FUNCTION_BLOCK FB_Encoder
VAR_INPUT
	nRawInput : UDINT;
	fEncoderOffset : LREAL; 
END_VAR
VAR_OUTPUT
	fPosition 		: LREAL;
	fPositionError 	: LREAL;
END_VAR
VAR PERSISTENT
	nRounds			: DINT;
	nRawLast 		: DINT;
END_VAR	
VAR
	nInput 		: DINT;
	nTempInputDiff	: DINT;
	nCount 			: DINT;
	nMaxValue30bit 	: DINT :=  1073741823; // 2^30 - 1	
	nThreshold30bit	: DINT := nMaxValue30bit/2;
	fScale16bit		: LREAL := 360.0/65535.0; // 360deg/(2^16 - 1)
	fTempPosition   : LREAL;
	fScaleDegtoMeter : LREAL := 0.075 * PI / 180 ; //Dette må endres senere, drum radius. 
	fPosRef 		 : LREAL;
END_VAR

// Convert to DINT (same as const values)
nInput := UDINT_TO_DINT(nRawInput);

// Define Encoder Rounds
nTempInputDiff := nInput - nRawLast;
IF (nTempInputDiff > nThreshold30bit) THEN
	nRounds := nRounds - 1;
END_IF

IF (nTempInputDiff < -nThreshold30bit) THEN
	nRounds := nRounds + 1;
END_IF

// Count Encoder Rounds
nCount := nInput + nRounds*nMaxValue30bit;

//Position Output
//fPosition := DINT_TO_LREAL(nCount)*fScale16bit - fEncoderOffset; // 

fPosition := (DINT_TO_LREAL(nCount)*fScale16bit - fEncoderOffset); //[deg]

END_FUNCTION_BLOCK

(* stored: Version 1.1.0.1, ProductVersion 3.1.4024.12
   POU FB_Encoder: Id {135b6917-e0f2-4f75-ba76-a6bf43c9c297}, SpecialFunc None *)
